PROGRAM POU_COM
VAR
	
END_VAR

//Instantiate COM 

(*Instanitate Serial port com function *) 

K4S8_DRL_03_E12_fbSerialLineControl(
	Mode:= SERIALLINEMODE_EL6_22B,
	pComIn:= ADR(K4S8_DRL_03_E12_stComIn),
	pComOut:=ADR(K4S8_DRL_03_E12_stComOut),
	SizeComIn:= SIZEOF(K4S8_DRL_03_E12_stComIn),
	TxBuffer:= K4S8_DRL_03_E12_EL6021_SerialTXBuffer,
	RxBuffer:= K4S8_DRL_03_E12_EL6021_SerialRXBuffer,
	Error=> ,
	ErrorID=> );

END_PROGRAM

(* stored: Version 1.1.0.1, ProductVersion 3.1.4022.18
   POU POU_COM: Id {d70bdf27-8797-4bac-87aa-9f251af83b06}, SpecialFunc None *)
